# EPICS autosave request: pluginsApp/Db/NDFitsN_settings.req
$(P)$(R)PeakAmplitude
$(P)$(R)PeakMu
$(P)$(R)PeakSigma
